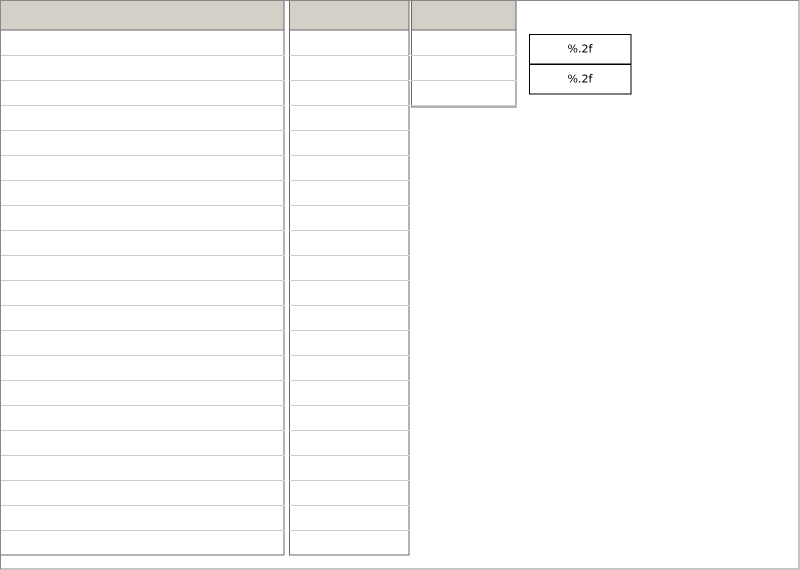
VISUALIZATION F99_IO_IO_2  // 800x570
    Table (0,0 284x555), data array: EL1809_S
        p3854506369: EL1809_S[1,INDEX]
        p1892666644: EL1809_S[2,INDEX]
        p338671338: EL1889_M[3,INDEX]
        Columns.Column.[1].Template: EL1809_S[2,INDEX]<>0
        Columns.Column.[0].Template: EL1809_S[1,INDEX]<>0
    Table (289,0 120x555), data array: EL2809_S
        p1892666644: EL2889_M[2,INDEX]
        p338671338: EL2889_M[3,INDEX]
        p2170511999: EL2889_M[4,INDEX]
        p3854506369: EL2809_S[1,INDEX]
        Columns.Column.[0].Template: EL2809_S[1,INDEX]<>0
    Table (411,0 105x107), data array: EL4002_S
        p3854506369: EL4002_S[INDEX]
    Rectangle (529,34 102x30), "%.2f", text variable: int_to_lreal(EL4002_S[1])/32767*10
    Rectangle (529,64 102x30), "%.2f", text variable: int_to_lreal(EL4002_S[2])/32767*10
END_VISUALIZATION

(* stored: Version 1.1.0.1, ProductVersion 3.1.4024.11
   Visu F99_IO_IO_2: Id {ece1d973-b755-4465-bc9c-92186d3cd21f} *)
